FUNCTION F_DT_ARG : ST_Arg
VAR_INPUT
	dtInput : DT;
END_VAR
VAR
	stArg : ST_Arg;
	sysVar_Info : __SYSTEM.VAR_INFO;
END_VAR

sysVar_Info 	:= __VARINFO(dtInput);
stArg.TypeClass := sysVar_Info.TypeClass;
stArg.pValue 	:= 0;
stArg.diSize 	:= SIZEOF(dtInput);
stArg.sValue 	:= TO_STRING(dtInput); 
THIS^ := stArg;

END_FUNCTION

(* stored: Version 1.1.0.1, ProductVersion 3.1.4024.4
   POU F_DT_ARG: Id {a4dadf69-c681-4af6-ac32-e10ead707b80}, SpecialFunc None *)
